(* IEC 61131-3 sources: repolevel_ST_code_completion/output/full_case_fixed/repoeval_Command1/readful_result, 11 files *)

(* ---- FB_AirConComfortCommand.st ---- *)
FUNCTION_BLOCK PUBLIC FB_AirConComfortCommand IMPLEMENTS I_Command
VAR
	refAirConditioning : REFERENCE TO FB_AirConditioning;
END_VAR

METHOD Execute : BOOL
VAR
  isValidRef : BOOL;
END_VAR

isValidRef := __ISVALIDREF(refAirConditioning);

IF isValidRef THEN
  refAirConditioning.Activate(); // Ensure this method exists in FB_AirConditioning
  refAirConditioning.SetTemperature(20.0); // Ensure SetTemperature(REAL) is defined in FB_AirConditioning
  Execute := TRUE;
ELSE
  Execute := FALSE;
END_IF
END_FUNCTION_BLOCK

(* ---- FB_AirConditioning.st ---- *)
FUNCTION_BLOCK PUBLIC FB_AirConditioning
VAR_OUTPUT
 bActive			: BOOL;
 lrTemperature	: LREAL;
END_VAR
VAR
 lrDefaultTemperature : LREAL := 22.0;
END_VAR

IF NOT bActive THEN
 lrTemperature := lrDefaultTemperature; // Explicitly set the output variable
ELSE
 lrTemperature := lrTemperature;        // Keep its value (already initialized externally if active)
END_IF

END_FUNCTION_BLOCK

(* ---- FB_AirConStandbyCommand.st ---- *)
FUNCTION_BLOCK PUBLIC FB_AirConStandbyCommand IMPLEMENTS I_Command
VAR
  refAirConditioning : REFERENCE TO FB_AirConditioning;
END_VAR

IF __ISVALIDREF(refAirConditioning) THEN
  refAirConditioning.bActive := FALSE;
END_IF
END_FUNCTION

(* ---- FB_CDPlayer.st ---- *)
FUNCTION_BLOCK PUBLIC FB_CDPlayer
VAR_OUTPUT
  bPlayerActive		: BOOL;
  byVolume			: BYTE;
  byTrack				: UINT;
END_VAR
VAR
  bInitialized : BOOL := FALSE;
END_VAR

IF NOT bInitialized THEN
 bPlayerActive := FALSE;
 byVolume := 50; // Default volume level
 byTrack := 1;   // Default track number
 bInitialized := TRUE;
END_IF

IF bPlayerActive THEN
  // Logic for active player state can be added here if needed
END_IF
END_FUNCTION_BLOCK

(* ---- FB_LampSetLevelCommand.st ---- *)
FUNCTION_BLOCK PUBLIC FB_LampSetLevelCommand IMPLEMENTS I_Command
VAR
refLamp		: REFERENCE TO FB_Lamp;
byNewLevel	: BYTE;
END_VAR

IF __ISVALIDREF(refLamp) THEN
refLamp.SetLevel(byNewLevel); // Check SetLevel implementation and refLamp initialization
END_IF
END_FUNCTION_BLOCK

(* ---- FB_MusicPlayCommand.st ---- *)
FUNCTION_BLOCK PUBLIC FB_MusicPlayCommand IMPLEMENTS I_Command
VAR
	refCDPlayer : REFERENCE TO FB_CDPlayer;
END_VAR

METHOD Execute

IF (__ISVALIDREF(THIS^.refCDPlayer)) THEN
// Ensure that the referenced object is valid and initialized
THIS^.refCDPlayer.SetVolume(40);
THIS^.refCDPlayer.SetTrack(1);
THIS^.refCDPlayer.Start();
ELSE
// Handle invalid reference case
// Placeholder for handling invalid references or initialization issues
END_IF
END_FUNCTION_BLOCK

(* ---- FB_MusicStopCommand.st ---- *)
FUNCTION_BLOCK PUBLIC FB_MusicStopCommand IMPLEMENTS I_Command
VAR
	refCDPlayer : REFERENCE TO FB_CDPlayer;
END_VAR

METHOD Execute

IF IS_VALID_REF(refCDPlayer) THEN
refCDPlayer.Stop();
END_IF
END_FUNCTION_BLOCK

(* ---- FB_Socket.st ---- *)
FUNCTION_BLOCK PUBLIC FB_Socket
VAR_OUTPUT
  bActive		: BOOL := FALSE;  // Ensure default output state
END_VAR
VAR
  bInitialized : BOOL := FALSE;
END_VAR

IF NOT bInitialized THEN
  bActive := FALSE;
  bInitialized := TRUE;
END_IF;
END_FUNCTION_BLOCK

(* ---- FB_SocketOffCommand.st ---- *)
FUNCTION_BLOCK PUBLIC FB_SocketOffCommand IMPLEMENTS I_Command
VAR
  refSocket : REFERENCE TO FB_Socket;
END_VAR

IF __ISVALIDREF(refSocket) THEN
  // Ensure refSocket is valid and that Off() is a callable method in FB_Socket
  refSocket^.Off();
END_IF
END_FUNCTION_BLOCK

(* ---- FB_SocketOnCommand.st ---- *)
FUNCTION_BLOCK PUBLIC FB_SocketOnCommand IMPLEMENTS I_Command
VAR
	refSocket : REFERENCE TO FB_Socket;
END_VAR

METHOD Execute
IF __ISVALIDREF(refSocket) THEN
 refSocket.On();
END_IF
RETURN;
END_FUNCTION_BLOCK

(* ---- FB_SwitchPanel.st ---- *)
FUNCTION_BLOCK PUBLIC FB_SwitchPanel
VAR_INPUT
	arrSwitch		: ARRAY[1..8] OF BOOL;
END_VAR
VAR
	aiCommand		: ARRAY[1..8] OF I_Command;
	arrRtrig		: ARRAY[1..8] OF R_TRIG;
	nIndex			: INT;
END_VAR

FOR nIndex := 1 TO 8 DO
  // Assign the `CLK` input of the R_TRIG function block
  arrRtrig[nIndex].CLK := arrSwitch[nIndex];
  IF arrRtrig[nIndex].Q THEN
    IF aiCommand[nIndex].Valid THEN
      aiCommand[nIndex].Execute();
    END_IF
  END_IF
END_FOR
END_FUNCTION_BLOCK
